FUNCTION F_ConvertTicksToUnixTimestamp : LREAL
VAR_INPUT
    nTimestamp : ULINT;
END_VAR
VAR CONSTANT
    // Timer ticks in Windows are 100ns (1e-7 sec)
    cfTicksToSeconds : LREAL := 10_000_000;
    // Epoch offset 1601 to 1970
    cfEpochOffset	: LREAL := 11_644_473_600;
END_VAR

F_ConvertTicksToUnixTimestamp := ULINT_TO_LREAL(nTimestamp) / cfTicksToSeconds - cfEpochOffset;

END_FUNCTION

(* stored: Version 1.1.0.1
   POU F_ConvertTicksToUnixTimestamp: Id {33156588-fcdd-4f41-9fa6-98babd8a3abc}, SpecialFunc None *)
